{attribute 'qualified_only'}
{attribute 'strict'}
{attribute 'to_string'}
TYPE E_SolenoidState :
(
	Open:=0, Closed:=1
);
END_TYPE

(* stored: Version 1.1.0.1
   DUT E_SolenoidState: Id {e39e76ff-5bbb-4e73-ab57-84d568312345} *)
